// TIA Portal V20 export
TYPE "LWONIK_typeSafetySensor"
// stored: Access Published
   STRUCT
      UnwinderLeftCartDetectSensor : Bool;
      UnwinderRightCartDetectSensor : Bool;
   END_STRUCT;
END_TYPE
